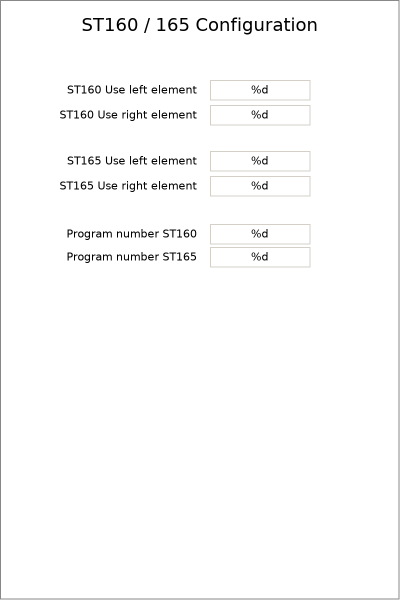
VISUALIZATION VISU_Recipe_ST160  // 400x600
    Textfield (210,80 100x20), "%d", text variable: _20_AUTO.recipe.st160.Use_element_left
        OnMouseDown: write the text variable via Default
    Label (0,5 400x40), "ST160 / 165 Configuration"
    Label (0,80 200x20), "ST160 Use left element"
    Textfield (210,105 100x20), "%d", text variable: _20_AUTO.recipe.st160.Use_element_right
        OnMouseDown: write the text variable via Default
    Label (0,105 200x20), "ST160 Use right element"
    Textfield (210,151 100x20), "%d", text variable: _20_AUTO.recipe.st165.Use_element_left
        OnMouseDown: write the text variable via Default
    Label (0,151 200x20), "ST165 Use left element"
    Textfield (210,176 100x20), "%d", text variable: _20_AUTO.recipe.st165.Use_element_right
        OnMouseDown: write the text variable via Default
    Label (0,176 200x20), "ST165 Use right element"
    Textfield (210,224 100x20), "%d", text variable: _20_AUTO.recipe.st160.Program_number
        OnMouseDown: write the text variable via Default
    Label (0,224 200x20), "Program number ST160"
    Textfield (210,247 100x20), "%d", text variable: _20_AUTO.recipe.st165.Program_number
        OnMouseDown: write the text variable via Default
    Label (0,247 200x20), "Program number ST165"
END_VISUALIZATION

(* stored: Version 1.1.0.1, ProductVersion 3.1.4024.6
   Visu VISU_Recipe_ST160: Id {cedf75af-695d-41a6-86be-517076040af4} *)
